FUNCTION_BLOCK L2_MachineState (* Basic Function Block Type *)
  (* Standard: 61499-2 *)
  (* Version 0.0, 2016-01-18, EQUEROL, UJI *)
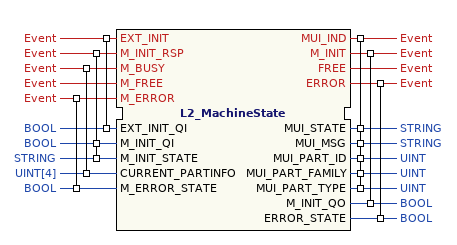
  EVENT_INPUT
    EXT_INIT WITH EXT_INIT_QI; (* Machine initialization Request *)
    M_INIT_RSP WITH M_INIT_QI, M_INIT_STATE; (* Machine initialization response *)
    M_BUSY WITH CURRENT_PARTINFO; (* Machine state changed to busy *)
    M_FREE; (* Machine state changed to free *)
    M_ERROR WITH M_ERROR_STATE; (* Machine state changed to error *)
  END_EVENT
  EVENT_OUTPUT
    MUI_IND WITH MUI_STATE, MUI_MSG, MUI_PART_ID, MUI_PART_FAMILY, MUI_PART_TYPE; (* MUI (Machine user inteface) indication *)
    M_INIT WITH M_INIT_QO; (* Machine initialization request *)
    FREE; (* Event to indicate L3 that the machine is free *)
    ERROR WITH ERROR_STATE; (* Event to indicate L3 that the machine is OK/KO *)
  END_EVENT
  VAR_INPUT
    EXT_INIT_QI : BOOL; (* Input event qualifier *)
    M_INIT_QI : BOOL; (* Machine initialization process qualifier *)
    M_INIT_STATE : STRING; (* String containing the state of the initialization process *)
    CURRENT_PARTINFO : ARRAY [0..3] OF UINT; (* Part's information of the new request *)
    M_ERROR_STATE : BOOL; (* Bool flag associated with M_ERROR event *)
  END_VAR
  VAR_OUTPUT
    MUI_STATE : STRING; (* String containing the state of the machine *)
    MUI_MSG : STRING; (* Message for the MUI containing information about machine's state *)
    MUI_PART_ID : UINT; (* Current part identifier *)
    MUI_PART_FAMILY : UINT; (* Current part family *)
    MUI_PART_TYPE : UINT; (* Current part type *)
    M_INIT_QO : BOOL; (* Machine initialization process qualifier *)
    ERROR_STATE : BOOL; (* Qualifier associated with error event *)
  END_VAR
  VAR
    initRequested : BOOL := FALSE; (* Flag to delay desinitilazitaion process until machine is idle *)
  END_VAR
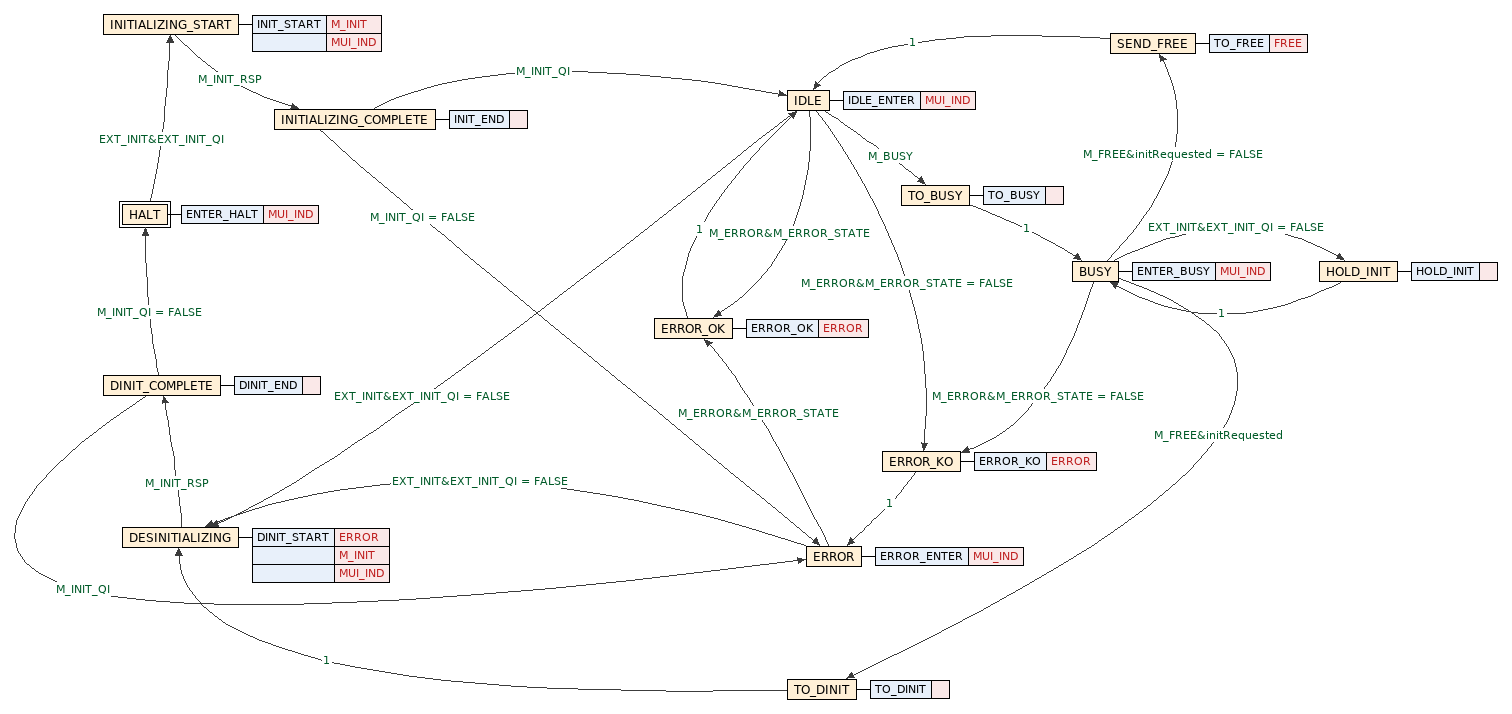
  EC_STATES
    HALT : ENTER_HALT -> MUI_IND;
    DESINITIALIZING : DINIT_START -> ERROR, -> M_INIT, -> MUI_IND;
    IDLE : IDLE_ENTER -> MUI_IND;
    BUSY : ENTER_BUSY -> MUI_IND;
    ERROR : ERROR_ENTER -> MUI_IND;
    INITIALIZING_COMPLETE : INIT_END;
    INITIALIZING_START : INIT_START -> M_INIT, -> MUI_IND;
    DINIT_COMPLETE : DINIT_END;
    SEND_FREE : TO_FREE -> FREE;
    ERROR_OK : ERROR_OK -> ERROR;
    ERROR_KO : ERROR_KO -> ERROR;
    HOLD_INIT : HOLD_INIT;
    TO_BUSY : TO_BUSY;
    TO_DINIT : TO_DINIT;
  END_STATES
  EC_TRANSITIONS
    INITIALIZING_COMPLETE TO IDLE := M_INIT_QI;
    INITIALIZING_COMPLETE TO ERROR := M_INIT_QI = FALSE;
    INITIALIZING_START TO INITIALIZING_COMPLETE := M_INIT_RSP;
    DESINITIALIZING TO DINIT_COMPLETE := M_INIT_RSP;
    DINIT_COMPLETE TO HALT := M_INIT_QI = FALSE;
    DINIT_COMPLETE TO ERROR := M_INIT_QI;
    HALT TO INITIALIZING_START := EXT_INIT&EXT_INIT_QI;
    ERROR TO DESINITIALIZING := EXT_INIT&EXT_INIT_QI = FALSE;
    IDLE TO DESINITIALIZING := EXT_INIT&EXT_INIT_QI = FALSE;
    BUSY TO SEND_FREE := M_FREE&initRequested = FALSE;
    SEND_FREE TO IDLE := 1;
    BUSY TO ERROR_KO := M_ERROR&M_ERROR_STATE = FALSE;
    IDLE TO ERROR_KO := M_ERROR&M_ERROR_STATE = FALSE;
    ERROR_KO TO ERROR := 1;
    ERROR TO ERROR_OK := M_ERROR&M_ERROR_STATE;
    ERROR_OK TO IDLE := 1;
    IDLE TO ERROR_OK := M_ERROR&M_ERROR_STATE;
    BUSY TO HOLD_INIT := EXT_INIT&EXT_INIT_QI = FALSE;
    HOLD_INIT TO BUSY := 1;
    IDLE TO TO_BUSY := M_BUSY;
    TO_BUSY TO BUSY := 1;
    BUSY TO TO_DINIT := M_FREE&initRequested;
    TO_DINIT TO DESINITIALIZING := 1;
  END_TRANSITIONS
  ALGORITHM INIT_START IN ST: (* Initialization algorithm *)
M_INIT_QO := TRUE;
MUI_STATE := "Initializing";
MUI_MSG := "Initializing machine...";
  END_ALGORITHM
  ALGORITHM INIT_END IN ST: (* new algorithm *)
MUI_MSG := M_INIT_STATE;
MUI_PART_ID:= 0;
MUI_PART_FAMILY := 0;
MUI_PART_TYPE := 0;
  END_ALGORITHM
  ALGORITHM IDLE_ENTER IN ST: (* new algorithm *)
MUI_STATE := "IDLE";
  END_ALGORITHM
  ALGORITHM ERROR_ENTER IN ST: (* new algorithm *)
MUI_STATE := "ERROR";
  END_ALGORITHM
  ALGORITHM DINIT_START IN ST: (* new algorithm *)
M_INIT_QO := FALSE;
MUI_STATE := "Desinitializing";
MUI_MSG := "Desinitializing machine...";
ERROR_STATE := FALSE;
  END_ALGORITHM
  ALGORITHM ENTER_HALT IN ST: (* new algorithm *)
MUI_STATE := "HALT";
  END_ALGORITHM
  ALGORITHM DINIT_END IN ST: (* new algorithm *)
MUI_MSG := M_INIT_STATE;
  END_ALGORITHM
  ALGORITHM ENTER_BUSY IN ST: (* new algorithm *)
MUI_STATE :="BUSY";
  END_ALGORITHM
  ALGORITHM ERROR_KO IN ST: (* new algorithm *)
ERROR_STATE := M_ERROR_STATE;
MUI_MSG := "An error occurred";
  END_ALGORITHM
  ALGORITHM HOLD_INIT IN ST: (* new algorithm *)
initRequested := TRUE;
MUI_MSG := "Desinitialization request registered";
  END_ALGORITHM
  ALGORITHM TO_FREE IN ST: (* new algorithm *)
MUI_MSG := "Part completed";
MUI_PART_ID:= 0;
MUI_PART_FAMILY := 0;
MUI_PART_TYPE := 0;
  END_ALGORITHM
  ALGORITHM ERROR_OK IN ST: (* new algorithm *)
ERROR_STATE := M_ERROR_STATE;
MUI_MSG := "Recovered from an error";
  END_ALGORITHM
  ALGORITHM TO_BUSY IN ST: (* new algorithm *)
MUI_MSG := "New part arrived";
MUI_PART_ID:= CURRENT_PARTINFO[0];
MUI_PART_FAMILY := CURRENT_PARTINFO[1];
MUI_PART_TYPE := CURRENT_PARTINFO[2];
  END_ALGORITHM
  ALGORITHM TO_DINIT IN ST: (* new algorithm *)
MUI_PART_ID:= 0;
MUI_PART_FAMILY := 0;
MUI_PART_TYPE := 0;
  END_ALGORITHM
END_FUNCTION_BLOCK
